// TIA Portal project "babu_TOFFusingTON" (V15)

(* hardware
DEVICE "S7-1200 station_1"  S7-1200 Station
   slot 0: "Rack_0"  S7-1200 Rack  Rack  V1.0
   slot 1: "PLC_1"  CPU 1212C DC/DC/DC  6ES7 212-1AE40-0XB0  V4.2
*)

// ===== PLC "PLC_1"  CPU 1212C DC/DC/DC =====

VAR_GLOBAL   // PLC tag table "Default tag table"
   "POWER ON" AT %M0.0 : Bool;
   "OUTPUT" AT %Q0.0 : Bool;
   "MEMORY" AT %M0.1 : Bool;
   "MEMORY OUTPUT" AT %M0.2 : Bool;
   "POWER ON TEST" AT %M0.3 : Bool;
   "OUTPUT 1" AT %Q0.1 : Bool;
END_VAR

// folder: System blocks/Program resources

DATA_BLOCK "IEC_Timer_0_DB"   // DB1
{ S7_Optimized_Access := 'TRUE' }
AUTHOR : Simatic
FAMILY : IEC
NAME : IEC_TMR
VERSION : 1.0
// stored: InstanceOfName IEC_TIMER
"IEC_TIMER"
BEGIN
END_DATA_BLOCK

DATA_BLOCK "IEC_Timer_0_DB_1"   // DB2
{ S7_Optimized_Access := 'TRUE' }
AUTHOR : Simatic
FAMILY : IEC
NAME : IEC_TMR
VERSION : 1.0
// stored: InstanceOfName IEC_TIMER
"IEC_TIMER"
BEGIN
END_DATA_BLOCK

// folder: (top level)

ORGANIZATION_BLOCK "Main"   // OB1, LAD, ProgramCycle
TITLE = "Main Program Sweep (Cycle)"
{ S7_Optimized_Access := 'TRUE' }
VERSION : 0.1
   VAR_INPUT
      Initial_Call : Bool;   // Initial call of this OB
      Remanence : Bool;   // =True, if remanent data are available
   END_VAR
BEGIN

REGION Network 1
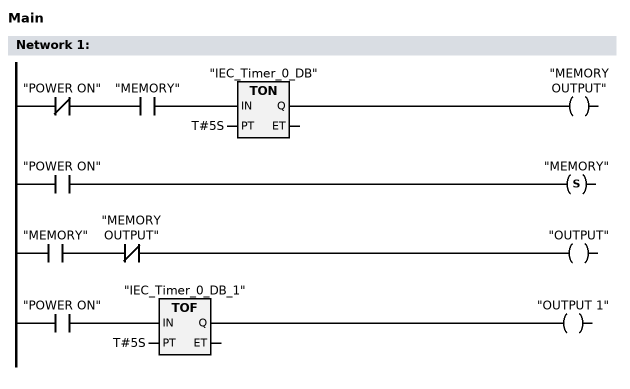
   "IEC_Timer_0_DB".TON(IN := NOT "POWER ON" AND "MEMORY", PT := T#5S);
   "MEMORY OUTPUT" := "IEC_Timer_0_DB".Q;
   IF "POWER ON" THEN "MEMORY" := TRUE; END_IF;
   "OUTPUT" := "MEMORY" AND NOT "MEMORY OUTPUT";
   "IEC_Timer_0_DB_1".TOF(IN := "POWER ON", PT := T#5S);
   "OUTPUT 1" := "IEC_Timer_0_DB_1".Q;
END_REGION
END_ORGANIZATION_BLOCK